Yaskawa INFORM job: MASTER_BATMAN_NEW_R1.JBI

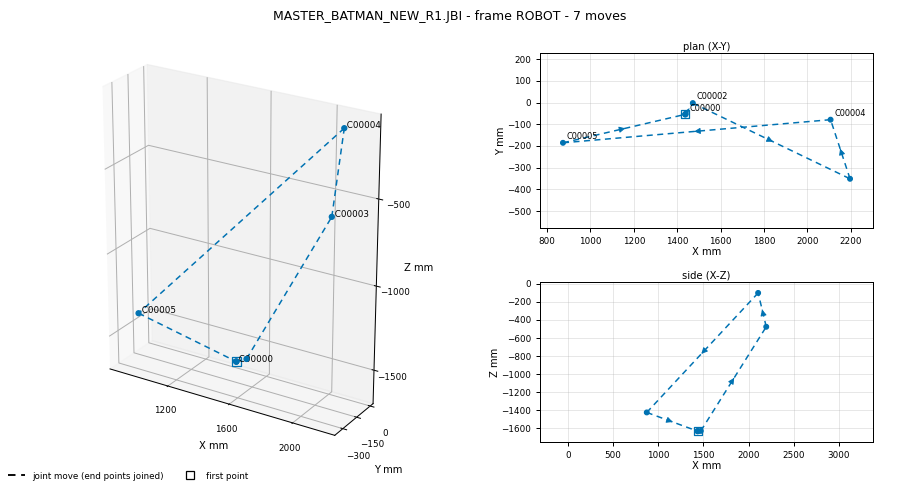
[picture p0: tool path of MASTER_BATMAN_NEW_R1.JBI in frame ROBOT, 7 of 7 moves have a stored position in this frame; points joined in program order, loops and branches not executed]
/JOB
//NAME MASTER_BATMAN_NEW_R1
///FOLDERNAME SCIANA_WYPYCHAJACA_V19B_V20
//POS
///NPOS 7,7,7,0,0,0
///TOOL 0
///POSTYPE ROBOT
///RECTAN
///RCONF 0,0,0,0,0,0,0,0,0,0,0,0,0,0,0,0,0,0,0,0,0,0,0,0
C00000=1437.133,-54.421,-1631.761,4.0165,22.0627,5.9438
///RCONF 0,0,0,0,1,0,0,0,0,0,0,0,0,0,0,0,0,0,0,0,0,0,0,0
C00001=1437.133,-54.420,-1631.761,4.0165,22.0627,5.9428
///RCONF 0,0,0,0,0,0,0,0,0,0,0,0,0,0,0,0,0,0,0,0,0,0,0,0
C00002=1471.732,-2.511,-1628.643,1.1536,25.5710,-67.1423
C00003=2196.406,-351.449,-475.392,-22.5516,45.7957,106.1638
///RCONF 0,0,0,0,1,0,0,0,0,0,0,0,0,0,0,0,0,0,0,0,0,0,0,0
C00004=2106.688,-78.970,-100.565,3.1885,-28.2868,5.2849
///RCONF 0,0,0,0,0,0,0,0,0,0,0,0,0,0,0,0,0,0,0,0,0,0,0,0
C00005=873.206,-185.580,-1423.876,-1.7383,27.7862,-167.3950
C00006=1437.133,-54.421,-1631.761,4.0165,22.0627,5.9438
BC00000=385.106,3798.155,1435.868
BC00001=385.106,3798.155,1538.047
BC00002=385.106,3798.155,1926.166
BC00003=411.619,32.863,1993.612
BC00004=176.597,1383.650,1999.736
BC00005=845.778,2972.171,1682.637
BC00006=385.106,3798.155,1435.868
///POSTYPE PULSE
///PULSE
EC00000=0,1
EC00001=-798157,-556476
EC00002=-798157,-556476
EC00003=-363194,-550745
EC00004=-798157,-556476
EC00005=-798157,-556476
EC00006=0,1
//INST
///DATE 2024/03/11 22:34
///ATTR SC,RW,RJ
////FRAME ROBOT
///GROUP1 RB1,BS1
///GROUP2 ST1
NOP
MOVJ C00000 BC00000 VJ=100.00  +MOVJ EC00000 VJ=100.00
MOVJ C00001 BC00001 VJ=100.00  +MOVJ EC00001 VJ=100.00
PAUSE
PAUSE
'SCIAGNIJ USZY ZE SCIANY
MOVJ C00002 BC00002 VJ=100.00  +MOVJ EC00002 VJ=100.00
MOVJ C00003 BC00003 VJ=100.00  +MOVJ EC00003 VJ=100.00
CALL JOB:BATMAN_ALL
MOVJ C00004 BC00004 VJ=50.00  +MOVJ EC00004 VJ=50.00
CALL JOB:BATMAN_2STR
MOVJ C00005 BC00005 VJ=50.00  +MOVJ EC00005 VJ=50.00
CALL JOB:BATMAN_4SPOINY
MOVJ C00006 BC00006 VJ=100.00  +MOVJ EC00006 VJ=100.00
PAUSE
END
